FUNCTION_BLOCK PULS_1S
VAR_INPUT
END_VAR
VAR_OUTPUT
	Q: BOOL;
END_VAR
VAR
	PULSO : BLINK;
END_VAR

PULSO(ENABLE:= TRUE, TIMELOW:= T#1S, TIMEHIGH:= T#1S, OUT=> Q);

END_FUNCTION_BLOCK

(* stored: Version 1.1.0.1, ProductVersion 3.1.4024.11
   POU PULS_1S: Id {19ea2cee-b869-4927-88e8-a6e83cc81e94}, SpecialFunc None *)
